PROGRAM MAIN
VAR
	fbTempModel : Temp_Model0;
	
	iVolt AT%I* : UINT;
	
	iTempSens1 AT%Q* : UINT;
	iTempSens2 AT%Q* : UINT;
	
END_VAR


fbTempModel(ssMethodType:= , iVolt_U:= iVolt , iTemp1_Y=> iTempSens1, iTemp2_Y=> iTempSens2 );
fbTempModel.ssMethodType := 1;

END_PROGRAM

(* stored: Version 1.1.0.1, ProductVersion 3.1.4024.13
   POU MAIN: Id {1f5639a3-112f-425f-8b43-e5799d7f7b16}, SpecialFunc None *)
